ABB RAPID module: Module1.mod

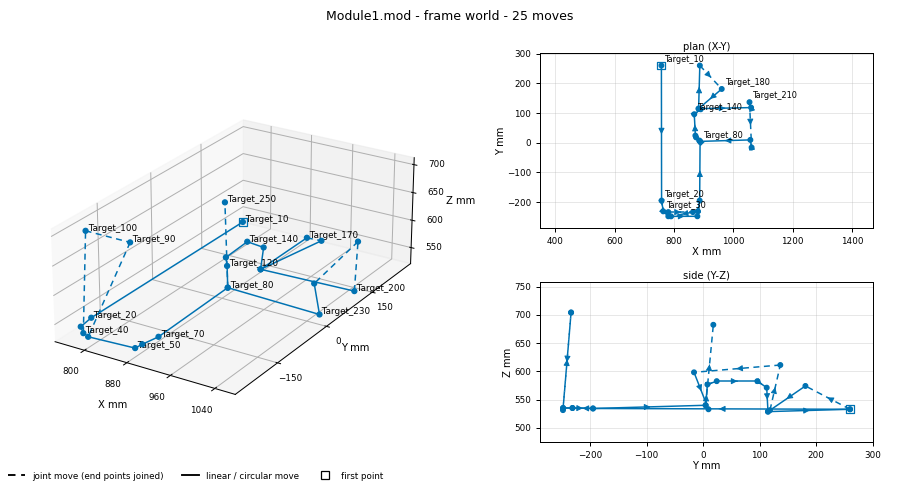
[picture p0: tool path of Module1.mod in frame world, 25 of 25 moves have a stored position in this frame; points joined in program order, loops and branches not executed]
MODULE Module1
        CONST robtarget Target_10:=[[0,60.271864372,14.72813562],[0.27059805,-0.653281482,-0.653281482,-0.27059805],[0,0,1,1],[9E+09,9E+09,9E+09,9E+09,9E+09,9E+09]];
    CONST robtarget Target_20:=[[455,60.857864372,16.14213562],[0.27059805,-0.653281482,-0.653281482,-0.27059805],[-1,-1,2,1],[9E+09,9E+09,9E+09,9E+09,9E+09,9E+09]];
    CONST robtarget Target_30:=[[491.351,66.582864372,16.97013562],[0.27059805,-0.653281482,-0.653281482,-0.27059805],[-1,-1,2,1],[9E+09,9E+09,9E+09,9E+09,9E+09,9E+09]];
    CONST robtarget Target_40:=[[507.970135761,83.530999911,16.970135486],[0.382683437,-0.000000001,-0.923879531,-0.000000002],[-1,-2,2,1],[9E+09,9E+09,9E+09,9E+09,9E+09,9E+09]];
    CONST robtarget Target_50:=[[507.970135761,181.468999911,16.970135486],[0.353553394,0.146446612,-0.85355339,0.353553388],[-1,0,0,0],[9E+09,9E+09,9E+09,9E+09,9E+09,9E+09]];
    CONST robtarget Target_60:=[[491.350999937,183.41713562,16.970135627],[0.14644661,0.353553391,-0.853553391,0.353553389],[-1,-1,0,0],[9E+09,9E+09,9E+09,9E+09,9E+09,9E+09]];
    CONST robtarget Target_70:=[[454.999999937,189.14213562,16.142135627],[0.146446612,0.353553391,-0.85355339,0.35355339],[-1,-1,0,0],[9E+09,9E+09,9E+09,9E+09,9E+09,9E+09]];
    CONST robtarget Target_80:=[[255.586000094,190.585999927,21.799203421],[0.353553392,0.353553392,-0.85355339,0.146446607],[-1,0,0,0],[9E+09,9E+09,9E+09,9E+09,9E+09,9E+09]];
    CONST robtarget Target_90:=[[493.828,166.469,186],[0.353553393,0.14644661,-0.853553388,0.353553395],[-1,0,0,0],[9E+09,9E+09,9E+09,9E+09,9E+09,9E+09]];
    CONST robtarget Target_100:=[[493.828,83.531,186],[0.382683433,0.000000004,-0.923879532,0.000000002],[-1,-2,-2,1],[9E+09,9E+09,9E+09,9E+09,9E+09,9E+09]];
    CONST robtarget Target_110:=[[508.184601642,92.798767036,13.220135652],[0.45710678,0.176776699,-0.85355339,0.176776696],[-1,0,0,0],[9E+09,9E+09,9E+09,9E+09,9E+09,9E+09]];
    CONST robtarget Target_120:=[[252.478469618,187.478122751,58.597199989],[0.353553392,0.353553392,-0.85355339,0.146446607],[-1,0,0,0],[9E+09,9E+09,9E+09,9E+09,9E+09,9E+09]];
    CONST robtarget Target_130:=[[236,174.751,64.5],[0,-0.707106781,0.707106782,0],[0,0,0,0],[9E+09,9E+09,9E+09,9E+09,9E+09,9E+09]];
    CONST robtarget Target_140:=[[163.999999997,171,64.5],[0,-0.707106781,0.707106782,0],[0,0,0,0],[9E+09,9E+09,9E+09,9E+09,9E+09,9E+09]];
    CONST robtarget Target_150:=[[147.500000005,192.677669427,53.00000015],[0.191341714,0.732537818,-0.461939767,0.461939764],[0,-1,-1,0],[9E+09,9E+09,9E+09,9E+09,9E+09,9E+09]];
    CONST robtarget Target_160:=[[145.271864442,185.58600014,10.585999953],[-0.000000004,0.70710678,-0.5,0.500000001],[0,-1,0,0],[9E+09,9E+09,9E+09,9E+09,9E+09,9E+09]];
    CONST robtarget Target_170:=[[0.000000011,189.72813562,14.728135627],[0.27059805,0.653281482,-0.653281483,0.27059805],[0,0,0,0],[9E+09,9E+09,9E+09,9E+09,9E+09,9E+09]];
    CONST robtarget Target_180:=[[79,263.5,56],[0.27059805,0.653281482,-0.653281483,0.27059805],[0,0,0,0],[9E+09,9E+09,9E+09,9E+09,9E+09,9E+09]];
    CONST robtarget Target_190:=[[145.271864442,185.58600014,10.585999953],[0.000000004,0.70710678,-0.5,0.500000001],[0,-1,0,0],[9E+09,9E+09,9E+09,9E+09,9E+09,9E+09]];
    CONST robtarget Target_200:=[[141.736330513,362.500000118,13.085999941],[0.000000004,0.70710678,-0.5,0.500000001],[0,-1,0,0],[9E+09,9E+09,9E+09,9E+09,9E+09,9E+09]];
    CONST robtarget Target_210:=[[123.423000005,357.07106781,93.071067814],[0.27059805,0.653281482,-0.653281483,0.27059805],[0,0,0,0],[9E+09,9E+09,9E+09,9E+09,9E+09,9E+09]];
    CONST robtarget Target_220:=[[276.201000011,364.14213562,80.142135627],[0.27059805,0.653281482,-0.653281483,0.27059805],[-1,-1,-1,0],[9E+09,9E+09,9E+09,9E+09,9E+09,9E+09]];
    CONST robtarget Target_230:=[[250.586000063,359.999999951,14.728135614],[0.353553392,0.353553392,-0.85355339,0.146446607],[0,0,0,0],[9E+09,9E+09,9E+09,9E+09,9E+09,9E+09]];
    CONST robtarget Target_240:=[[255.586000094,190.585999927,21.799203421],[0.353553392,0.353553392,-0.85355339,0.146446607],[0,0,0,0],[9E+09,9E+09,9E+09,9E+09,9E+09,9E+09]];
    CONST robtarget Target_250:=[[242.00000014,176.999999889,164.284271247],[0.353553392,0.353553392,-0.85355339,0.146446607],[0,0,0,0],[9E+09,9E+09,9E+09,9E+09,9E+09,9E+09]];
    CONST robtarget Target_260:=[[150.955000003,188.187135542,53.094000119],[0.191341714,0.732537818,-0.461939767,0.461939764],[0,-1,-1,0],[9E+09,9E+09,9E+09,9E+09,9E+09,9E+09]];
!***********************************************************
    !
    ! Module:  Module1
    !
    ! Description:
    !   <Insert description here>
    !
    ! Author: ASUS
    !
    ! Version: 1.0
    !
    !***********************************************************


    !***********************************************************
    !
    ! Procedure main
    !
    !   This is the entry point of your program
    !
    !***********************************************************

    PROC Path_10()
        MoveJ Target_10,v150,z0,Gorionik\WObj:=wobj_ploca;
        MoveL Target_20,v100,z0,Gorionik\WObj:=wobj_ploca;
        MoveL Target_30,v100,z0,Gorionik\WObj:=wobj_ploca;
        MoveL Target_40,v100,z0,Gorionik\WObj:=wobj_ploca;
        MoveJ Target_100,v150,z10,Gorionik\WObj:=wobj_ploca;
        MoveJ Target_90,v200,z10,Gorionik\WObj:=wobj_ploca;
        MoveJ Target_110,v150,z10,Gorionik\WObj:=wobj_ploca;
        MoveL Target_50,v100,z0,Gorionik\WObj:=wobj_ploca;
        MoveL Target_60,v100,z0,Gorionik\WObj:=wobj_ploca;
        MoveL Target_70,v100,z0,Gorionik\WObj:=wobj_ploca;
        MoveL Target_80,v100,z0,Gorionik\WObj:=wobj_ploca;
        MoveL Target_120,v100,z0,Gorionik\WObj:=wobj_ploca;
        MoveL Target_130,v100,z0,Gorionik\WObj:=wobj_ploca;
        MoveL Target_140,v100,z0,Gorionik\WObj:=wobj_ploca;
        MoveL Target_150,v100,z0,Gorionik\WObj:=wobj_ploca;
        MoveL Target_160,v100,z0,Gorionik\WObj:=wobj_ploca;
        MoveL Target_170,v100,z0,Gorionik\WObj:=wobj_ploca;
        MoveJ Target_180,v150,z0,Gorionik\WObj:=wobj_ploca;
        MoveL Target_190,v100,z0,Gorionik\WObj:=wobj_ploca;
        MoveL Target_200,v100,z0,Gorionik\WObj:=wobj_ploca;
        MoveJ Target_210,v150,z10,Gorionik\WObj:=wobj_ploca;
        MoveJ Target_220,v150,z10,Gorionik\WObj:=wobj_ploca;
        MoveL Target_230,v100,z0,Gorionik\WObj:=wobj_ploca;
        MoveL Target_240,v100,z0,Gorionik\WObj:=wobj_ploca;
        MoveJ Target_250,v150,z10,Gorionik\WObj:=wobj_ploca;
    ENDPROC
    PROC main_1()
        Path_10;
    ENDPROC
    PROC main()
        Path_10;
    ENDPROC
ENDMODULE
